// TwinCAT 3 PLC project PLC
// ProgramVersion: 3.1.4023.0
// libraries:
//   Tc2_Standard, * (Beckhoff Automation GmbH)
//   Tc2_System, * (Beckhoff Automation GmbH)
//   Tc3_IoLink, * (Beckhoff Automation GmbH)
//   Tc3_Module, * (Beckhoff Automation GmbH)
// project tree:
//   / PlcTask.TcTTO
//   POUs/ FB_IO_Link_Festo.TcPOU, FB_Read_IoLinkSpecs.TcPOU, Festo_IoLink_VacumEjector_OVEM_H_CE.TcPOU, MAIN.TcPOU
// real-time tasks:
//   TASK PlcTask: cycle T#10ms, priority 20, ADS port 350
// I/O:
//   DEVICE Device 1 (EtherCAT), AmsNetId 5.24.130.144.2.1
//     Term 1 (EK1200) [EK1200-5000 EtherCAT Power supply (2A E-Bus)]
//       Term 4 (EL1008) [EL1008 8Ch. Dig. Input 24V, 3ms]
//       Term 2 (EL6224) [EL6224 (IO Link Master)]
//       Term 3 (EL9011) [EL9011 End Terminal]
// variable links:
//   PLC Instance <-> Device 1 (EtherCAT)/Term 1 (EK1200)/Term 2 (EL6224)
//     PlcTask Inputs/MAIN.amsNetId <-> InfoData/AoeNetId
//     PlcTask Inputs/MAIN.pressure <-> IO-Link Port1_in/Pressure value

CONFIGURATION PLC
    RESOURCE PLC ON TwinCAT3
        TASK PlcTask(INTERVAL := T#10ms, PRIORITY := 20);
        PROGRAM MAIN WITH PlcTask : MAIN;
    END_RESOURCE
END_CONFIGURATION

// ---- POUs/MAIN.TcPOU
PROGRAM MAIN
VAR
     Festo           : Festo_IoLink_VacumEjector_OVEM_H_CE;
     Execute         : BOOL;
     amsNetId AT %I* : AMSNETID;
     netid    AT %I* : T_AmsNetId;

     Port AT %I* : UINT;

     pressure AT %I* : UINT;
END_VAR

IO_Link();

ACTION IO_Link:
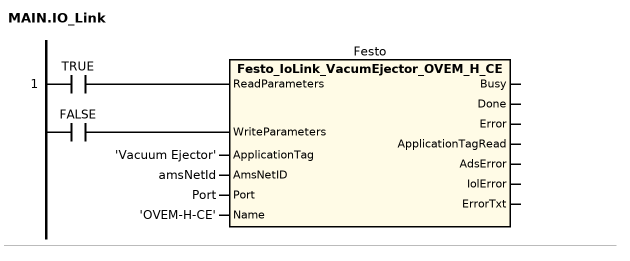
// NETWORK 1
Festo(
    ReadParameters := TRUE,
    WriteParameters := FALSE,
    ApplicationTag := 'Vacuum Ejector',
    AmsNetID := amsNetId,
    Port := Port,
    Name := 'OVEM-H-CE'); // Festo_IoLink_VacumEjector_OVEM_H_CE
END_ACTION

END_PROGRAM

// ---- POUs/Festo_IoLink_VacumEjector_OVEM_H_CE.TcPOU
FUNCTION_BLOCK Festo_IoLink_VacumEjector_OVEM_H_CE
VAR_INPUT
     ReadParameters  : BOOL;             // Read parameters
     WriteParameters : BOOL;             // Set parameters
     Reset           : BOOL;             // Reset application 
     ApplicationTag  : STRING(32) := ''; // Application Tag 
     AmsNetID        : AMSNETID;         // AMS Net ID 
     Port            : UINT;             // Port on IO link terminal 
     Name            : STRING(255);      // Name of IO link device
END_VAR
VAR_OUTPUT
     Busy               : BOOL       := FALSE;
     Done               : BOOL       := FALSE;
     Error              : BOOL       := FALSE;
     ApplicationTagRead : STRING(32) := '';
     AirSaveFunction    : BOOL;
     AutoDropTime       : INT; // 0x0198 - 80 
     AdsError           : E_AdsErr    := E_AdsErr.NOERR;
     IolError           : E_IolError  := E_IolError.NoError;
     ErrorTxt           : STRING(255) := '';
END_VAR
VAR
     _InitDone           : BOOL := FALSE;
     _ReadParameters     : BOOL; // Read parameters
     _SetParameters      : BOOL; // Set parameters
     _ApplicationTagRead : STRING(32) := '';
     _ReadState          : INT        := 0;
     _SetState           : INT        := 0;
     _fbIolSlave         : FB_IolStdVarSlave;
     _fbIolVarSlave      : FB_IolSlave;
     _hr                 : HRESULT;
     Start               : BOOL;

     _State : INT; // case state	

     _rtReadParameter  : R_TRIG;
     _rtWriteParameter : R_TRIG;

END_VAR

_rtReadParameter(CLK := ReadParameters);
_rtWriteParameter(CLK := WriteParameters);

CASE _State OF

     00: //Init 
          _InitDone                  := TRUE;
          _fbIolSlave.MasterAoeNetId := F_CreateAmsNetId(AmsNetID); //Creates NETID String
          _fbIolSlave.Port           := Port;
          _fbIolSlave.Name           := Name;
          _State                     := 10;

     10: // Idle

          IF _rtReadParameter.Q THEN
               _State := 20;
          ELSIF _rtWriteParameter.Q THEN
               _State := 120;
          END_IF

     20: // Read Parameters 
          // Read Application Tag

          _hr := _fbIolSlave.ReadApplicationSpecificTag(ApplicationTagRead);

          IF NOT F_IolIsBusy(_hr) THEN
               IF FAILED(_hr) THEN
                    Busy       := FALSE;
                    Error      := TRUE;
                    ErrorTxt   := _fbIolSlave.ErrorTxt; // TODO
                    AdsError   := F_IolGetAdsError(_hr);
                    IolError   := F_IolGetIolError(_hr);
                    _ReadState := 999; // Error;
               ELSE
                    _ReadState := 30; // CHECK;
               END_IF
          END_IF
		30: // Read



     999: // Error state 

          IF Reset THEN
               Busy     := FALSE;
               Error    := FALSE;
               AdsError := E_AdsErr.NOERR;
               IolError := E_IolError.NoError;
               ErrorTxt := '';
          END_IF
END_CASE

METHOD PRIVATE ReadApplicationTag : UDINT
VAR_INPUT 
	Execute : BOOL; 
END_VAR
////
// FB State Machine
//
CASE _ReadState OF

     // IDLE
     0: ;

          IF Execute THEN
               _ReadState := 10;
          END_IF

     10: // Read application Tag

          _hr := _fbIolSlave.ReadApplicationSpecificTag(ApplicationTagRead);

          IF NOT F_IolIsBusy(_hr) THEN
               IF FAILED(_hr) THEN
                    Busy       := FALSE;
                    Error      := TRUE;
                    ErrorTxt   := _fbIolSlave.ErrorTxt; // TODO
                    AdsError   := F_IolGetAdsError(_hr);
                    IolError   := F_IolGetIolError(_hr);
                    _ReadState := 999; // Error;
               ELSE
                    _ReadState := 30; // CHECK;
               END_IF
          END_IF

     // CHECK
     30: IF ApplicationTag <> _ApplicationTagRead THEN
               Busy     := FALSE;
               Error    := TRUE;
               ErrorTxt := 'sApplicationTag and sApplicationTagRead are not equal!';
          ELSE
               Busy := FALSE;
               Done := TRUE;
               //              _ReadState := 0;
          END_IF

     999: // Error state

          IF NOT Execute THEN

               _hr := _fbIolSlave.SysCmdApplicationReset();

               IF NOT F_IolIsBusy(_hr) THEN
                    IF FAILED(_hr) THEN
                         Busy     := FALSE;
                         Error    := TRUE;
                         ErrorTxt := _fbIolSlave.ErrorTxt; 
                         AdsError := F_IolGetAdsError(_hr);
                         IolError := F_IolGetIolError(_hr);
                         //_ReadState := 999; // Error;
                    ELSE
                         _ReadState := 0; // CHECK;
                    END_IF
               END_IF

          END_IF

END_CASE

////
// call FBs
//
_fbIolSlave();
END_METHOD

METHOD PRIVATE WriteApplicationTag : UDINT
VAR_INPUT
END_VAR
END_METHOD

END_FUNCTION_BLOCK

// ---- POUs/FB_IO_Link_Festo.TcPOU
FUNCTION_BLOCK FB_IO_Link_Festo
VAR_INPUT
     bExecute        : BOOL       := FALSE;
     sApplicationTag : STRING(32) := '';
     sAmsNetID       : STRING;
     Port            : UINT;
     Name            : STRING;
END_VAR
VAR_OUTPUT
     bBusy     : BOOL        := FALSE;
     bDone     : BOOL        := FALSE;
     bError    : BOOL        := FALSE;
     nAdsError : E_AdsErr    := E_AdsErr.NOERR;
     nIolError : E_IolError  := E_IolError.NoError;
     sErrorTxt : STRING(255) := '';
END_VAR
VAR
     bInitDone           : BOOL := FALSE;
     bExecuteOld         : BOOL;
     nState              : INT := 0;
     sApplicationTagRead : STRING(32) := '';
     fbIolSlave          : FB_IolSlave;
     hr                  : HRESULT;

END_VAR

////
// Init
//
IF NOT bInitDone THEN
     bInitDone                 := TRUE;
     fbIolSlave.MasterAoeNetId := F_CreateAmsNetId(sAmsNetID);
     fbIolSlave.Port           := Port;
     fbIolSlave.Name           := Name;
END_IF

////
// Execute/Busy State Machine
//
IF bExecute AND NOT bExecuteOld AND NOT bBusy THEN
     bBusy  := TRUE;
     nState := 10; // WRITE
ELSIF NOT bExecute THEN
     bBusy     := FALSE;
     bError    := FALSE;
     bDone     := FALSE;
     nAdsError := E_AdsErr.NOERR;
     nIolError := E_IolError.NoError;
     sErrorTxt := '';
END_IF

bExecuteOld := bExecute;

////
// FB State Machine
//
CASE nState OF

     // IDLE
     0: ;

     // WRITE
     10: hr := fbIolSlave.Write(16#0018,
                                0,
                                ADR(sApplicationTag),
                                INT_TO_UDINT(LEN(sApplicationTag)));

          IF NOT F_IolIsBusy(hr) THEN
               IF FAILED(hr) THEN
                    bBusy     := FALSE;
                    bError    := TRUE;
                    sErrorTxt := fbIolSlave.ErrorTxt; // TODO
                    nAdsError := F_IolGetAdsError(hr);
                    nIolError := F_IolGetIolError(hr);
                    nState    := 0; // IDLE;
               ELSE
                    nState := 20; // WRITE;
               END_IF
          END_IF

     // READ
     20: hr := fbIolSlave.Read(16#0018,
                               16#00,
                               ADR(sApplicationTagRead),
                               SIZEOF(sApplicationTagRead));

          IF NOT F_IolIsBusy(hr) THEN
               IF FAILED(hr) THEN
                    bBusy     := FALSE;
                    bError    := TRUE;
                    sErrorTxt := fbIolSlave.ErrorTxt; // TODO
                    nAdsError := F_IolGetAdsError(hr);
                    nIolError := F_IolGetIolError(hr);
                    nState    := 0; // IDLE;
               ELSE
                    nState := 30; // CHECK;
               END_IF
          END_IF

     // CHECK
     30: IF sApplicationTag <> sApplicationTagRead THEN
               bBusy     := FALSE;
               bError    := TRUE;
               sErrorTxt := 'sApplicationTag and sApplicationTagRead are not equal!';
          ELSE
               bBusy  := FALSE;
               bDone  := TRUE;
               nState := 0;
          END_IF
END_CASE

////
// call FBs
//
fbIolSlave();

END_FUNCTION_BLOCK

// ---- POUs/FB_Read_IoLinkSpecs.TcPOU
FUNCTION_BLOCK FB_Read_IoLinkSpecs
VAR_INPUT
     bExecute        : BOOL       := FALSE;
     sApplicationTag : STRING(32) := '';
     sAmsNetID       : STRING;
     Port            : UINT;
     Name            : STRING(255);

END_VAR
VAR_OUTPUT
     bBusy     : BOOL        := FALSE;
     bDone     : BOOL        := FALSE;
     bError    : BOOL        := FALSE;
     nAdsError : E_AdsErr    := E_AdsErr.NOERR;
     nIolError : E_IolError  := E_IolError.NoError;
     sErrorTxt : STRING(255) := '';
END_VAR
VAR
     bExecuteOld         : BOOL;
     nState              : INT := 0;
     fbIolVarSlave          : FB_IolStdVarSlave;
     bInitDone           : BOOL := FALSE;
     hr                  : HRESULT;
     sApplicationTagRead : STRING(32) := '';
END_VAR

////
// Init
//
IF NOT bInitDone THEN
     bInitDone                 := TRUE;
     fbIolVarSlave.MasterAoeNetId := F_CreateAmsNetId(sAmsNetID); //Creates NETID String
     fbIolVarSlave.Port           := Port;
     fbIolVarSlave.Name           := Name;
END_IF

////
// Execute/Busy State Machine
//
IF bExecute AND NOT bExecuteOld AND NOT bBusy THEN
     bBusy  := TRUE;
     nState := 10; // WRITE
ELSIF NOT bExecute THEN
     bBusy     := FALSE;
     bError    := FALSE;
     bDone     := FALSE;
     nAdsError := E_AdsErr.NOERR;
     nIolError := E_IolError.NoError;
     sErrorTxt := '';
END_IF

bExecuteOld := bExecute;

////
// FB State Machine
//
CASE nState OF

     // IDLE
     0: ;

     // WRITE
     10: hr := fbIolVarSlave.WriteApplicationSpecificTag(sApplicationTag);

          IF NOT F_IolIsBusy(hr) THEN
               IF FAILED(hr) THEN
                    bBusy     := FALSE;
                    bError    := TRUE;
                    sErrorTxt := fbIolVarSlave.ErrorTxt; // TODO
                    nAdsError := F_IolGetAdsError(hr);
                    nIolError := F_IolGetIolError(hr);
                    nState    := 0; // IDLE;
               ELSE
                    nState := 20; // WRITE;
               END_IF
          END_IF

     // READ
     20: hr := fbIolVarSlave.ReadApplicationSpecificTag(sApplicationTagRead);

          IF NOT F_IolIsBusy(hr) THEN
               IF FAILED(hr) THEN
                    bBusy     := FALSE;
                    bError    := TRUE;
                    sErrorTxt := fbIolVarSlave.ErrorTxt; // TODO
                    nAdsError := F_IolGetAdsError(hr);
                    nIolError := F_IolGetIolError(hr);
                    nState    := 0; // IDLE;
               ELSE
                    nState := 30; // CHECK;
               END_IF
          END_IF

     // CHECK
     30: IF sApplicationTag <> sApplicationTagRead THEN
               bBusy     := FALSE;
               bError    := TRUE;
               sErrorTxt := 'sApplicationTag and sApplicationTagRead are not equal!';
          ELSE
               bBusy  := FALSE;
               bDone  := TRUE;
               nState := 0;
          END_IF
END_CASE

////
// call FBs
//
fbIolVarSlave();

END_FUNCTION_BLOCK
